% RSLogix 500 project rev_pulse_masks.RSS, saved by version 8.30.00.16 %
PROJECT "UNTITLED"    % processor: Bul.1763 MicroLogix 1100 Series B %

PROGRAM FILES
  LAD 2   6 rungs

DATA FILES
  O0 OUTPUT  4 elements
  I1 INPUT  6 elements
  S2 STATUS  66 elements
  B3 BINARY  24 elements
  T4 TIMER  1 elements
  C5 COUNTER  1 elements
  R6 CONTROL  1 elements
  N7 INTEGER  2 elements
  F8 FLOAT  10 elements
  L9 MISCELLANY  10 elements
  L20 ONE_BITS  24 elements  % 1,2,4,8,10,20,... %
  L21 LOW_MASKS  24 elements  % 0,1,3,7,F,1F,3F,... %

LADDER 2
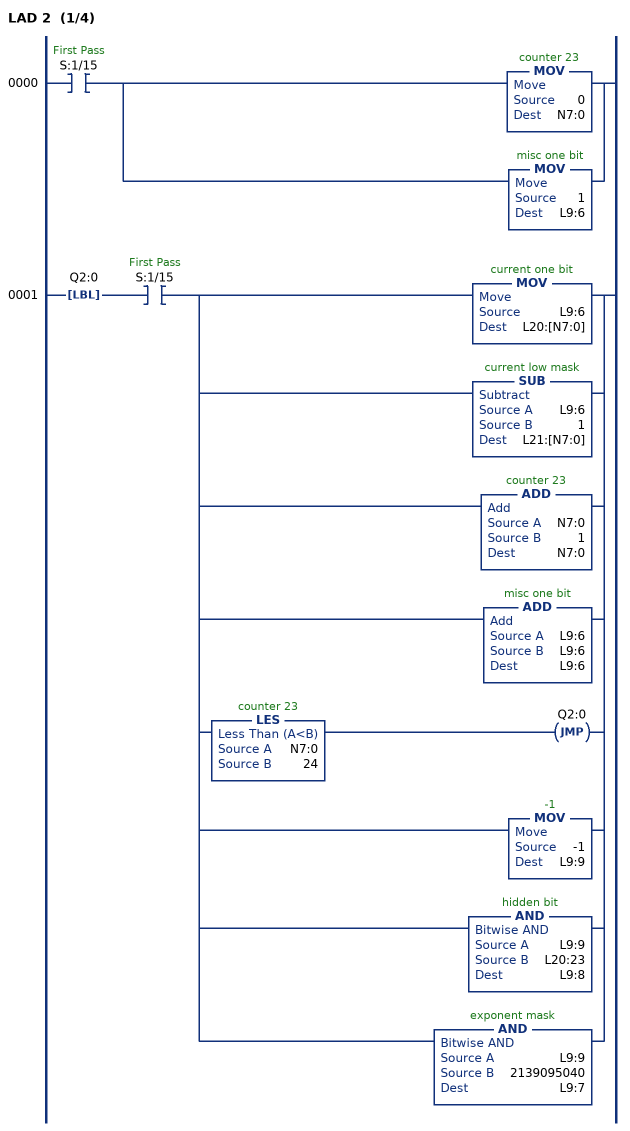
% Rung: 0 %
SOR XIC S:1/15 BST MOV 0 N7:0 NXB MOV 1 L9:6 BND EOR
%   S:1/15  "First Pass" %
%   N7:0  "counter 23" %
%   L9:6  "misc one bit" %
% Rung: 1 %
SOR LBL Q2:0 XIC S:1/15 BST MOV L9:6 L20:[N7:0] NXB SUB L9:6 1 L21:[N7:0] NXB ADD N7:0 1 N7:0 NXB ADD L9:6 L9:6 L9:6 NXB LES N7:0 24 JMP Q2:0 NXB MOV -1 L9:9 NXB AND L9:9 L20:23 L9:8 NXB AND L9:9 2139095040 L9:7 BND EOR
%   S:1/15  "First Pass" %
%   L9:6  "misc one bit" %
%   L20:[N7:0]  "current one bit" %
%   N7:0  "counter 23" %
%   L21:[N7:0]  "current low mask" %
%   L9:9  "-1" %
%   L9:8  "hidden bit" %
%   L9:7  "exponent mask" %

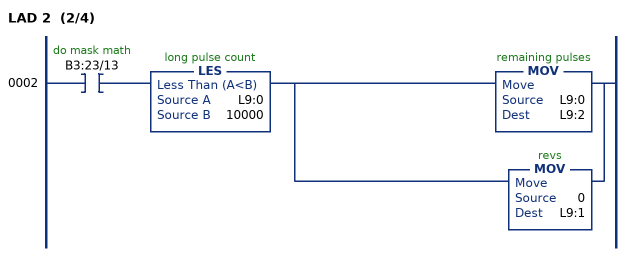
% Rung: 2 %
SOR XIC B3:23/13 LES L9:0 10000 BST MOV L9:0 L9:2 NXB MOV 0 L9:1 BND EOR
%   B3:23/13  "do mask math" %
%   L9:0  "long pulse count" %
%   L9:2  "remaining pulses" %
%   L9:1  "revs" %

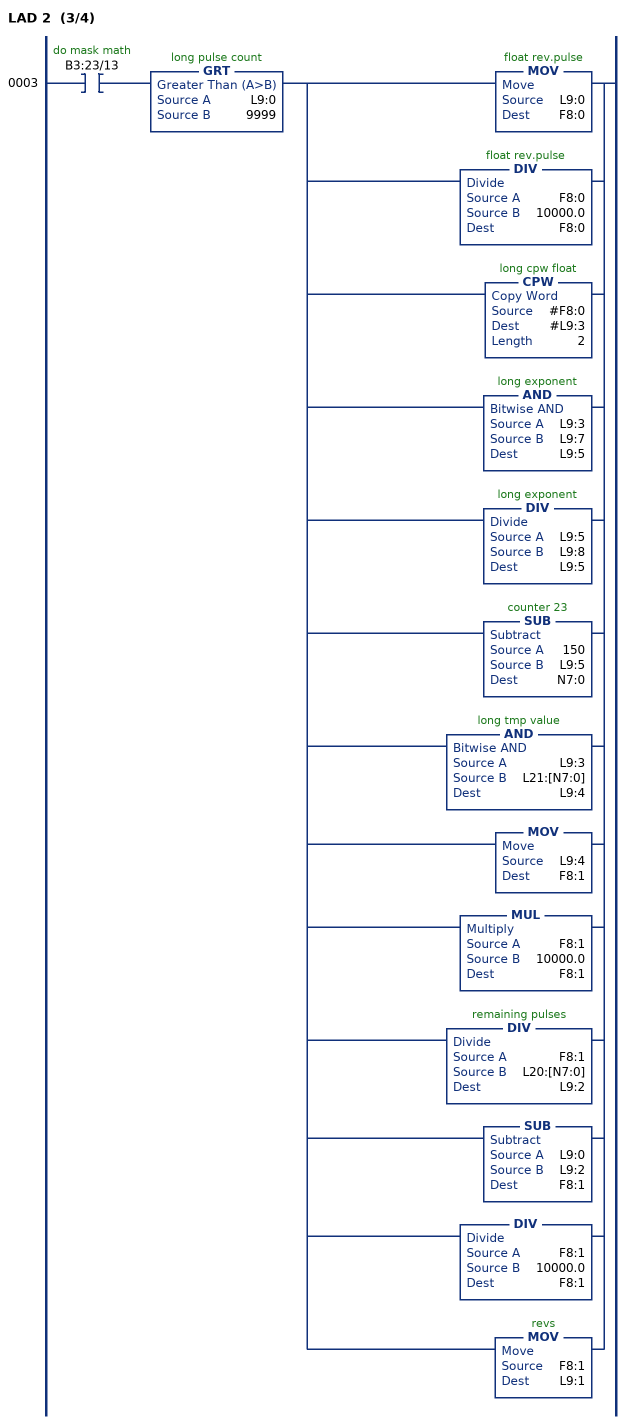
% Rung: 3 %
SOR XIC B3:23/13 GRT L9:0 9999 BST MOV L9:0 F8:0 NXB DIV F8:0 10000.0 F8:0 NXB CPW #F8:0 #L9:3 2 NXB AND L9:3 L9:7 L9:5 NXB DIV L9:5 L9:8 L9:5 NXB SUB 150 L9:5 N7:0 NXB AND L9:3 L21:[N7:0] L9:4 NXB MOV L9:4 F8:1 NXB MUL F8:1 10000.0 F8:1 NXB DIV F8:1 L20:[N7:0] L9:2 NXB SUB L9:0 L9:2 F8:1 NXB DIV F8:1 10000.0 F8:1 NXB MOV F8:1 L9:1 BND EOR
%   B3:23/13  "do mask math" %
%   L9:0  "long pulse count" %
%   F8:0  "float rev.pulse" %
%   L9:3  "long cpw float" %
%   L9:7  "exponent mask" %
%   L9:5  "long exponent" %
%   L9:8  "hidden bit" %
%   N7:0  "counter 23" %
%   L21:[N7:0]  "current low mask" %
%   L9:4  "long tmp value" %
%   L20:[N7:0]  "current one bit" %
%   L9:2  "remaining pulses" %
%   L9:1  "revs" %

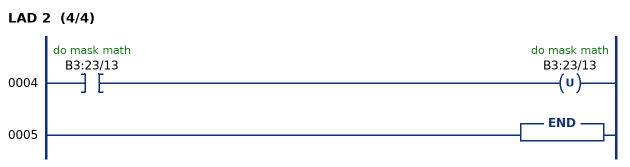
% Rung: 4 %
SOR XIC B3:23/13 OTU B3:23/13 EOR
%   B3:23/13  "do mask math" %
% Rung: 5 %
SOR END EOR
